FUNCTION_BLOCK FB_DetectorFotoelectrico EXTENDS FB_Module
(*

ESTACIONES DE DETECCIÓN DE MATERIAL - Manual de usuario #32/28

Con el fin de diferenciar finalmente las tapas de nylon blanco de las de
color negro, se ha incluido un detector fotoeléctrico. Dicho componente 
proporciona una señal de detección únicamente, de las tapas de color 
blanco
 
*)

VAR_OUTPUT
	// Controlador
   	fbController: FB_Simple_SFC:=(dr:=dr);

	// Sensores
    df         : dvSensor := (dr:=dr); //AT %I*: BOOL; (* ef  (nombre=df  c=I32 B=J1 b=04 módulo=EL1008 T=7  C=7 etiqueta=-B20, input) Detector fotoeléctrico *)

	Lectura_Registrada: BOOL := FALSE; 
	Tapa_Clara: BOOL;
	strUi : STRING := '?';
END_VAR

METHOD ProcessCycle : BOOL
VAR_INPUT
	dr			: REFERENCE TO FB_Director;
	tapas		: REFERENCE TO FB_Tapas;	
END_VAR
// Pause y reset
IsStopped := NOT fbController.UnsafeStop AND (dr.gmModeActual = E_GEMMA.A3ParadaEstado);
fbController.SFCReset := dr.gmModeActual = E_GEMMA.A6Inicializando;
fbController.SFCPause := IsStopped;

df.ProcessCycle(dr:=dr);
IC := InitialConditions();
fbController(
	dr:=dr, IC:=IC, Execute:=Execute, Ack:=Ack, Ready=>Ready, Done=>Done);

IF Done AND NOT Lectura_Registrada THEN
	// si ha terminado de captar: guardar resultado
	Lectura_Registrada	:= TRUE;
	Tapa_Clara			:= df.uiValue;
	strUi := SEL(Tapa_Clara, 'Oscura','Clara');
	tapas.Claridad(Tapa_Clara:=Tapa_Clara);
ELSIF Ready THEN
	// una vez que cambia el ciclo la lectura ya no es fiable
	Lectura_Registrada		:= FALSE;
	strUi := '?';
END_IF
END_METHOD

END_FUNCTION_BLOCK

(* stored: Version 1.1.0.1, ProductVersion 3.1.4024.11
   POU FB_DetectorFotoelectrico: Id {9c6b326b-8120-4a79-942a-3ee0b68cb66a}, SpecialFunc None
   Method ProcessCycle: Id {357ca19b-a2f2-4f95-9ae5-44e396b69f2c} *)
